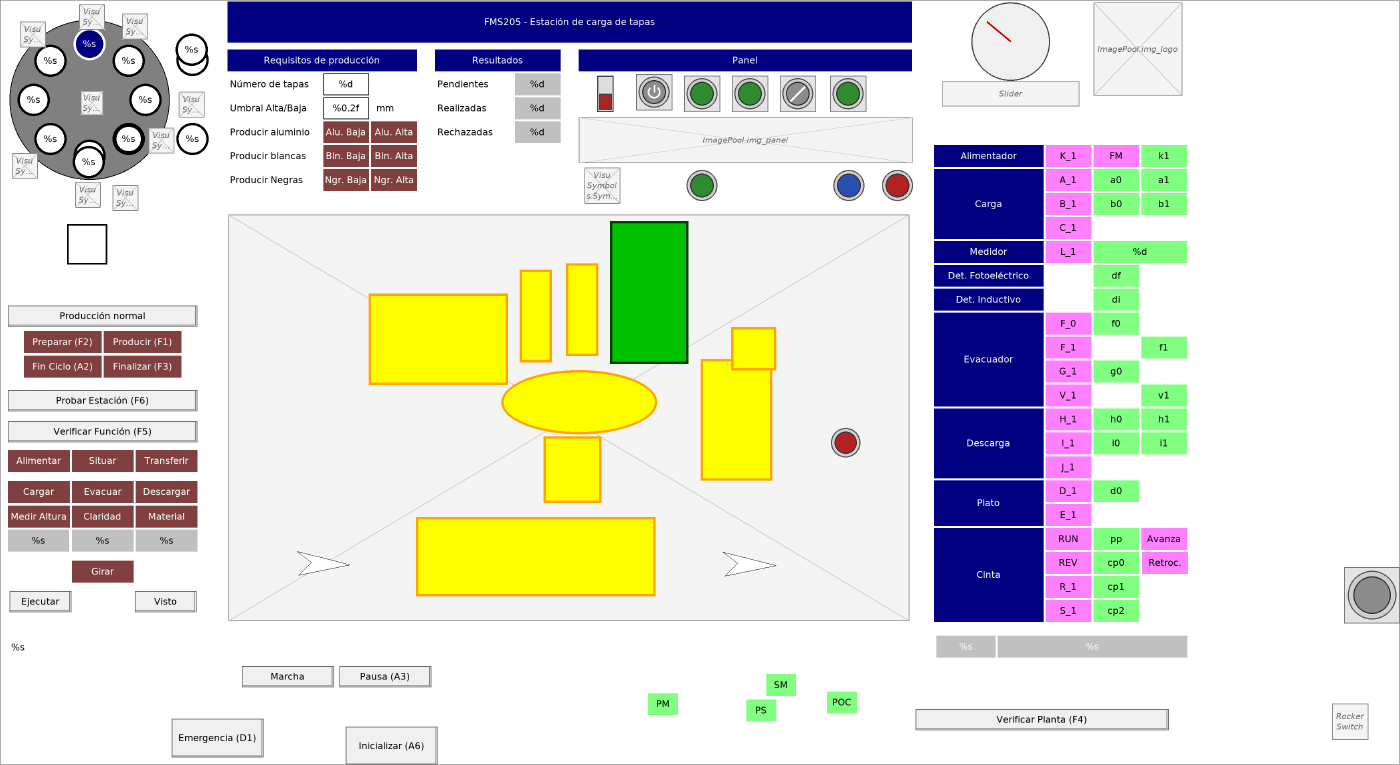
VISUALIZATION L5_FMS205VISU  // 1754x959
    Rectangle (285,2 857x51), "FMS205 - Estación de carga de tapas", colour variable: MAIN.fbFMS205.dr.gmModeColor
        p3450524324: MAIN.fbFMS205.dr.gmModeColor
    Rectangle (285,62 237x27), "Requisitos de producción"
    Rectangle (545,62 157x27), "Resultados"
    Rectangle (725,62 417x27), "Panel"
    Rectangle (285,92 157x27), "Número de tapas"
    Rectangle (405,92 57x27), "%d", text variable: MAIN.fbFMS205.tapas.ReqNumero
        OnMouseClick: write the text variable via VisuDialogs.Numpad, min 1, max 500
    Rectangle (545,92 97x27), "Pendientes"
    Rectangle (645,92 57x27), "%d", text variable: MAIN.fbFMS205.tapas.ResPend
    Rectangle (1036,867 37x27), "POC", input disabled if: NOT MAIN.fbFMS205.dr.gmLocalHost
        toggle MAIN.fbFMS205.fbPanel.hwPOC_PulsadorReset
    Rectangle (812,869 37x27), "PM", input disabled if: NOT MAIN.fbFMS205.dr.gmLocalHost
        toggle MAIN.fbFMS205.fbPanel.hwPM_PulsadorMarcha
    Rectangle (960,845 37x27), "SM", input disabled if: NOT MAIN.fbFMS205.dr.gmLocalHost
        toggle MAIN.fbFMS205.fbPanel.hwSM_SelecAutoManual
    Rectangle (285,122 117x27), "Umbral Alta/Baja"
    Rectangle (405,122 57x27), "%0.2f", text variable: MAIN.fbFMS205.tapas.ReqAlta
        p4168582468: 'Atura en mm mínima para considerar que la tapa es alta'
        OnMouseClick: write the text variable via VisuDialogs.Numpad, min 2, max 5
    Rectangle (465,122 37x27), "mm"
    Rectangle (545,122 117x27), "Realizadas"
    Rectangle (645,122 57x27), "%d", text variable: MAIN.fbFMS205.tapas.ResReal
    Rectangle (285,152 117x27), "Producir aluminio"
    Rectangle (405,152 57x27), "Alu. Baja"
        toggle MAIN.fbFMS205.tapas.ReqAluBaja
    Rectangle (465,152 57x27), "Alu. Alta"
        toggle MAIN.fbFMS205.tapas.ReqAluAlta
    Rectangle (545,152 117x27), "Rechazadas"
    Rectangle (645,152 57x27), "%d", text variable: MAIN.fbFMS205.tapas.ResRech
    Button (1147,889 317x26), "Verificar Planta (F4)", tooltip "%s"
        toggle MAIN.fbFMS205.fbPanel.mdF4Planta
    Rectangle (285,182 117x27), "Producir blancas"
    Rectangle (405,182 57x27), "Bln. Baja"
        toggle MAIN.fbFMS205.tapas.ReqBlnBaja
    Rectangle (465,182 57x27), "Bln. Alta"
        toggle MAIN.fbFMS205.tapas.ReqBlnAlta
    Rectangle (1170,182 137x27), "Alimentador", input disabled if: not MAIN.fbFMS205.dr.cnF4_Planta
    Rectangle (1310,182 57x27), "K_1", input disabled if: not MAIN.fbFMS205.dr.cnF4_Planta
        toggle MAIN.fbFMS205.mdAlimentador.K_1.uiValue
    Rectangle (1370,182 57x27), "FM", input disabled if: not MAIN.fbFMS205.dr.cnF4_Planta
        toggle MAIN.fbFMS205.mdAlimentador.FM.uiValue
    Rectangle (1430,182 57x27), "k1", input disabled if: not MAIN.fbFMS205.dr.cnF4_Planta
        toggle MAIN.fbFMS205.mdAlimentador.k1.uiValue
    Rectangle (285,212 117x27), "Producir Negras"
    Rectangle (405,212 57x27), "Ngr. Baja"
        toggle MAIN.fbFMS205.tapas.ReqNgrBaja
    Rectangle (465,212 57x27), "Ngr. Alta"
        toggle MAIN.fbFMS205.tapas.ReqNgrAlta
    Rectangle (1170,212 137x87), "Carga", input disabled if: not MAIN.fbFMS205.dr.cnF4_Planta
    Rectangle (1310,212 57x27), "A_1", input disabled if: not MAIN.fbFMS205.dr.cnF4_Planta
        toggle MAIN.fbFMS205.mdPickAndPlaceCarga.HOR.uiValue
    Rectangle (1370,212 57x27), "a0", input disabled if: not MAIN.fbFMS205.dr.cnF4_Planta
        toggle MAIN.fbFMS205.mdPickAndPlaceCarga.h0.uiValue
    Rectangle (1430,212 57x27), "a1", input disabled if: not MAIN.fbFMS205.dr.cnF4_Planta
        toggle MAIN.fbFMS205.mdPickAndPlaceCarga.h1.uiValue
    Rectangle (1310,242 57x27), "B_1", input disabled if: not MAIN.fbFMS205.dr.cnF4_Planta
        toggle MAIN.fbFMS205.mdPickAndPlaceCarga.VER.uiValue
    Rectangle (1370,242 57x27), "b0", input disabled if: not MAIN.fbFMS205.dr.cnF4_Planta
        toggle MAIN.fbFMS205.mdPickAndPlaceCarga.v0.uiValue
    Rectangle (1430,242 57x27), "b1", input disabled if: not MAIN.fbFMS205.dr.cnF4_Planta
        toggle MAIN.fbFMS205.mdPickAndPlaceCarga.v1.uiValue
    Rectangle (286,269 837x507), "Estacion"
    Button (303,835 115x26), "Marcha"
        tap MAIN.fbFMS205.fbPanel.swF0_Empezar
    Rectangle (30,415 97x27), "Preparar (F2)", input disabled if: not MAIN.fbFMS205.fbPanel.mdF1Producir
        toggle MAIN.fbFMS205.fbPanel.swF2_Preparar
    Rectangle (130,415 97x27), "Producir (F1)", input disabled if: not MAIN.fbFMS205.fbPanel.mdF1Producir
        toggle MAIN.fbFMS205.fbPanel.swF1_Producir
    Button (215,901 115x48), "Emergencia (D1)", tooltip "%s"
        p4168582468: MAIN.fbFMS205.fbPanel.ttPE_Seta
        toggle MAIN.fbFMS205.fbPanel.swPE_Seta
    Button (425,835 115x26), "Pausa (A3)"
        tap MAIN.fbFMS205.fbPanel.swA3_Estado
    Rectangle (1310,272 57x27), "C_1", input disabled if: not MAIN.fbFMS205.dr.cnF4_Planta
        toggle MAIN.fbFMS205.mdPickAndPlaceCarga.PIN.uiValue
    Rectangle (1170,302 137x27), "Medidor", input disabled if: not MAIN.fbFMS205.dr.cnF4_Planta
    Rectangle (1310,302 57x27), "L_1", input disabled if: not MAIN.fbFMS205.dr.cnF4_Planta
        toggle MAIN.fbFMS205.mdMedidorTapa.L_1.uiValue
    Rectangle (1370,302 117x27), "%d", text variable: MAIN.fbFMS205.mdMedidorTapa.dh, input disabled if: not MAIN.fbFMS205.dr.cnF4_Planta
    Rectangle (1170,332 137x27), "Det. Fotoeléctrico", input disabled if: not MAIN.fbFMS205.dr.cnF4_Planta
    Rectangle (1370,332 57x27), "df", input disabled if: not MAIN.fbFMS205.dr.cnF4_Planta
        toggle MAIN.fbFMS205.mdDetectorFotoelectrico.df.uiValue
    Rectangle (1170,362 137x27), "Det. Inductivo", input disabled if: not MAIN.fbFMS205.dr.cnF4_Planta
    Rectangle (1370,362 57x27), "di", input disabled if: not MAIN.fbFMS205.dr.cnF4_Planta
        toggle MAIN.fbFMS205.mdCaptadorInductivo.di.uiValue
    Rectangle (1170,392 137x117), "Evacuador", input disabled if: not MAIN.fbFMS205.dr.cnF4_Planta
    Rectangle (1310,392 57x27), "F_0", input disabled if: not MAIN.fbFMS205.dr.cnF4_Planta
        toggle MAIN.fbFMS205.mdEvacuador.F_0.uiValue
    Rectangle (1370,392 57x27), "f0", input disabled if: not MAIN.fbFMS205.dr.cnF4_Planta
        toggle MAIN.fbFMS205.mdEvacuador.f0.uiValue
    Button (10,528 237x26), "Verificar Función (F5)", input disabled if: not (MAIN.fbFMS205.dr.gmModeActual=L1_GEMMA.F5VerificacionOrdenada or MAIN.fbFMS205.dr.gmModeActual=L1_GEMMA.A1ParadaInicial)
        toggle MAIN.fbFMS205.fbPanel.mdF5Funcion
    Rectangle (1310,422 57x27), "F_1", input disabled if: not MAIN.fbFMS205.dr.cnF4_Planta
        toggle MAIN.fbFMS205.mdEvacuador.F_1.uiValue
    Rectangle (1430,422 57x27), "f1", input disabled if: not MAIN.fbFMS205.dr.cnF4_Planta
        toggle MAIN.fbFMS205.mdEvacuador.f1.uiValue
    Rectangle (10,564 77x27), "Alimentar", input disabled if: MAIN.fbFMS205.dr.gmModeActual<>L1_GEMMA.F5VerificacionOrdenada
        toggle MAIN.fbFMS205.fbPanel.swF5_Alimentar
    Rectangle (90,703 77x27), "Girar", input disabled if: MAIN.fbFMS205.dr.gmModeActual<>L1_GEMMA.F5VerificacionOrdenada
        toggle MAIN.fbFMS205.fbPanel.swF5_Girar
    Rectangle (90,564 77x27), "Situar", input disabled if: MAIN.fbFMS205.dr.gmModeActual<>L1_GEMMA.F5VerificacionOrdenada
        toggle MAIN.fbFMS205.fbPanel.swF5_Situar
    Rectangle (10,634 77x27), "Medir Altura", input disabled if: MAIN.fbFMS205.dr.gmModeActual<>L1_GEMMA.F5VerificacionOrdenada
        toggle MAIN.fbFMS205.fbPanel.swF5_Medir
    Rectangle (90,634 77x27), "Claridad", input disabled if: MAIN.fbFMS205.dr.gmModeActual<>L1_GEMMA.F5VerificacionOrdenada
        toggle MAIN.fbFMS205.fbPanel.swF5_Claridad
    Rectangle (170,634 77x27), "Material", input disabled if: MAIN.fbFMS205.dr.gmModeActual<>L1_GEMMA.F5VerificacionOrdenada
        toggle MAIN.fbFMS205.fbPanel.swF5_Material
    Rectangle (10,664 76x27), "%s", text variable: MAIN.fbFMS205.mdMedidorTapa.strUi, input disabled if: MAIN.fbFMS205.dr.gmModeActual<>L1_GEMMA.F5VerificacionOrdenada
    Rectangle (90,664 77x27), "%s", text variable: MAIN.fbFMS205.mdDetectorFotoelectrico.strUi, input disabled if: MAIN.fbFMS205.dr.gmModeActual<>L1_GEMMA.F5VerificacionOrdenada
    Rectangle (170,664 77x27), "%s", text variable: MAIN.fbFMS205.mdCaptadorInductivo.strUi, input disabled if: MAIN.fbFMS205.dr.gmModeActual<>L1_GEMMA.F5VerificacionOrdenada
    Rectangle (10,603 77x27), "Cargar", input disabled if: MAIN.fbFMS205.dr.gmModeActual<>L1_GEMMA.F5VerificacionOrdenada
        toggle MAIN.fbFMS205.fbPanel.swF5_Cargar
    Rectangle (90,603 77x27), "Evacuar", input disabled if: MAIN.fbFMS205.dr.gmModeActual<>L1_GEMMA.F5VerificacionOrdenada
        toggle MAIN.fbFMS205.fbPanel.swF5_Evacuar
    Rectangle (170,603 77x27), "Descargar", input disabled if: MAIN.fbFMS205.dr.gmModeActual<>L1_GEMMA.F5VerificacionOrdenada
        toggle MAIN.fbFMS205.fbPanel.swF5_Descargar
    Rectangle (170,564 77x27), "Transferir", input disabled if: MAIN.fbFMS205.dr.gmModeActual<>L1_GEMMA.F5VerificacionOrdenada
        toggle MAIN.fbFMS205.fbPanel.swF5_Transferir
    Button (12,741 77x26), "Ejecutar", input disabled if: MAIN.fbFMS205.dr.gmModeActual<>L1_GEMMA.F5VerificacionOrdenada
        tap MAIN.fbFMS205.fbPanel.swF5_Ejecutar
    Button (169,741 77x26), "Visto", input disabled if: MAIN.fbFMS205.dr.gmModeActual<>L1_GEMMA.F5VerificacionOrdenada
        tap MAIN.fbFMS205.fbPanel.swF5_Ack
    Rectangle (1310,452 57x27), "G_1", input disabled if: not MAIN.fbFMS205.dr.cnF4_Planta
        toggle MAIN.fbFMS205.mdEvacuador.G_1.uiValue
    Rectangle (1370,452 57x27), "g0", input disabled if: not MAIN.fbFMS205.dr.cnF4_Planta
        toggle MAIN.fbFMS205.mdEvacuador.g0.uiValue
    Rectangle (1310,482 57x27), "V_1", input disabled if: not MAIN.fbFMS205.dr.cnF4_Planta
        toggle MAIN.fbFMS205.mdEvacuador.V_1.uiValue
    Rectangle (1430,482 57x27), "v1", input disabled if: not MAIN.fbFMS205.dr.cnF4_Planta
        toggle MAIN.fbFMS205.mdEvacuador.v1.uiValue
    Rectangle (1170,512 137x87), "Descarga", input disabled if: not MAIN.fbFMS205.dr.cnF4_Planta
    Rectangle (1310,512 57x27), "H_1", input disabled if: not MAIN.fbFMS205.dr.cnF4_Planta
        toggle MAIN.fbFMS205.mdPickAndPlaceDescarga.HOR.uiValue
    Rectangle (1370,512 57x27), "h0", input disabled if: not MAIN.fbFMS205.dr.cnF4_Planta
        tap MAIN.fbFMS205.mdPickAndPlaceDescarga.h0.uiValue
        toggle MAIN.fbFMS205.mdPickAndPlaceDescarga.h0.uiValue
    Rectangle (1430,512 57x27), "h1", input disabled if: not MAIN.fbFMS205.dr.cnF4_Planta
        toggle MAIN.fbFMS205.mdPickAndPlaceDescarga.h1.uiValue
    Rectangle (1310,542 57x27), "I_1", input disabled if: not MAIN.fbFMS205.dr.cnF4_Planta
        toggle MAIN.fbFMS205.mdPickAndPlaceDescarga.VER.uiValue
    Rectangle (1370,542 57x27), "i0", input disabled if: not MAIN.fbFMS205.dr.cnF4_Planta
        toggle MAIN.fbFMS205.mdPickAndPlaceDescarga.v0.uiValue
    Rectangle (1430,542 57x27), "i1", input disabled if: not MAIN.fbFMS205.dr.cnF4_Planta
        toggle MAIN.fbFMS205.mdPickAndPlaceDescarga.v1.uiValue
    Rectangle (1310,572 57x27), "J_1", input disabled if: not MAIN.fbFMS205.dr.cnF4_Planta
        toggle MAIN.fbFMS205.mdPickAndPlaceDescarga.PIN.uiValue
    Rectangle (1170,602 137x57), "Plato", input disabled if: not MAIN.fbFMS205.dr.cnF4_Planta
    Rectangle (1310,602 57x27), "D_1", input disabled if: not MAIN.fbFMS205.dr.cnF4_Planta
        toggle MAIN.fbFMS205.mdPlatoDivisor.D_1.uiValue
    Rectangle (1370,602 57x27), "d0", input disabled if: not MAIN.fbFMS205.dr.cnF4_Planta
        toggle MAIN.fbFMS205.mdPlatoDivisor.d0.uiValue
    Rectangle (1310,632 57x27), "E_1", input disabled if: not MAIN.fbFMS205.dr.cnF4_Planta
        toggle MAIN.fbFMS205.mdPlatoDivisor.E_1.uiValue
    Rectangle (1170,662 137x117), "Cinta", input disabled if: not MAIN.fbFMS205.dr.cnF4_Planta
    Rectangle (1310,662 57x27), "RUN", input disabled if: not MAIN.fbFMS205.dr.cnF4_Planta
        toggle MAIN.fbFMS205.mdCinta.RUN.uiValue
    Rectangle (1370,662 57x27), "pp", input disabled if: not MAIN.fbFMS205.dr.cnF4_Planta
        toggle MAIN.fbFMS205.mdCinta.pp.uiValue
    Rectangle (1430,662 57x27), "Avanza", colour toggle: MAIN.fbFMS205.mdCinta.RUN.uiValue and Not MAIN.fbFMS205.mdCinta.REV.uiValue, input disabled if: not MAIN.fbFMS205.dr.cnF4_Planta
        tap MAIN.fbFMS205.fbPanel.swF4_Avanza
    Rectangle (1310,692 57x27), "REV", input disabled if: not MAIN.fbFMS205.dr.cnF4_Planta
        toggle MAIN.fbFMS205.mdCinta.REV.uiValue
    Rectangle (1370,692 57x27), "cp0", input disabled if: not MAIN.fbFMS205.dr.cnF4_Planta
        toggle MAIN.fbFMS205.mdCinta.cp0.uiValue
    Rectangle (1431,692 57x27), "Retroc.", colour toggle: MAIN.fbFMS205.mdCinta.RUN.uiValue and MAIN.fbFMS205.mdCinta.REV.uiValue, input disabled if: not MAIN.fbFMS205.dr.cnF4_Planta
        tap MAIN.fbFMS205.fbPanel.swF4_Retroc
    Rectangle (1310,722 57x27), "R_1", input disabled if: not MAIN.fbFMS205.dr.cnF4_Planta
        toggle MAIN.fbFMS205.mdCinta.R_1.uiValue
    Rectangle (1370,722 57x27), "cp1", input disabled if: not MAIN.fbFMS205.dr.cnF4_Planta
        toggle MAIN.fbFMS205.mdCinta.cp1.uiValue
    Rectangle (1310,752 57x27), "S_1", input disabled if: not MAIN.fbFMS205.dr.cnF4_Planta
        toggle MAIN.fbFMS205.mdCinta.S_1.uiValue
    Rectangle (1370,752 57x27), "cp2", input disabled if: not MAIN.fbFMS205.dr.cnF4_Planta
        toggle MAIN.fbFMS205.mdCinta.cp2.uiValue
    Rectangle (11,798 1117x27), "%s", text variable: main.fbFMS205.fbPanel.swMensaje
    Rectangle (1173,797 74x27), "%s", text variable: MAIN.fbFMS205.fbPanel.gmModeName, colour variable: MAIN.fbFMS205.dr.gmModeColor
        p3450524324: MAIN.fbFMS205.dr.gmModeColor
    Rectangle (1250,797 237x27), "%s", text variable: MAIN.fbFMS205.fbPanel.gmModeDescr, colour variable: MAIN.fbFMS205.dr.gmModeColor
        p3450524324: MAIN.fbFMS205.dr.gmModeColor
    Ellipse (12,25 200x200), colour variable: colVacFrameSin
        p3450524324: colVacFill
    Ellipse (162,105 40x40), "%s", tooltip "%s", text variable: MAIN.fbFMS205.tapas.vstrUi[7], colour variable: MAIN.fbFMS205.tapas.vColorFill[7]
        p2277200375: MAIN.fbFMS205.mdPlatoDivisor.Angulo
        p4168582468: MAIN.fbFMS205.tapas.vstrToolTip[7]
        p55702900: MAIN.fbFMS205.tapas.vColorFont[7]
        p3450524324: MAIN.fbFMS205.tapas.vColorFrame[7]
    Ellipse (141,154 40x40), "%s", tooltip "%s", text variable: MAIN.fbFMS205.tapas.vstrUi[0], colour variable: MAIN.fbFMS205.tapas.vColorFill[0]
        p2277200375: MAIN.fbFMS205.mdPlatoDivisor.Angulo
        p4168582468: MAIN.fbFMS205.tapas.vstrToolTip[0]
        p55702900: MAIN.fbFMS205.tapas.vColorFont[0]
        p3450524324: MAIN.fbFMS205.tapas.vColorFrame[0]
    Ellipse (92,175 40x40), "%s", tooltip "%s", text variable: MAIN.fbFMS205.tapas.vstrUi[1], colour variable: MAIN.fbFMS205.tapas.vColorFill[1]
        p2277200375: MAIN.fbFMS205.mdPlatoDivisor.Angulo
        p4168582468: MAIN.fbFMS205.tapas.vstrToolTip[1]
        p55702900: MAIN.fbFMS205.tapas.vColorFont[1]
        p3450524324: MAIN.fbFMS205.tapas.vColorFrame[1]
    Ellipse (43,154 40x40), "%s", tooltip "%s", text variable: MAIN.fbFMS205.tapas.vstrUi[2], colour variable: MAIN.fbFMS205.tapas.vColorFill[2]
        p2277200375: MAIN.fbFMS205.mdPlatoDivisor.Angulo
        p4168582468: MAIN.fbFMS205.tapas.vstrToolTip[2]
        p55702900: MAIN.fbFMS205.tapas.vColorFont[2]
        p3450524324: MAIN.fbFMS205.tapas.vColorFrame[2]
    Ellipse (22,105 40x40), "%s", tooltip "%s", text variable: MAIN.fbFMS205.tapas.vstrUi[3], colour variable: MAIN.fbFMS205.tapas.vColorFill[3]
        p2277200375: MAIN.fbFMS205.mdPlatoDivisor.Angulo
        p4168582468: MAIN.fbFMS205.tapas.vstrToolTip[3]
        p55702900: MAIN.fbFMS205.tapas.vColorFont[3]
        p3450524324: MAIN.fbFMS205.tapas.vColorFrame[3]
    Ellipse (43,56 40x40), "%s", tooltip "%s", text variable: MAIN.fbFMS205.tapas.vstrUi[4], colour variable: MAIN.fbFMS205.tapas.vColorFill[4]
        p2277200375: MAIN.fbFMS205.mdPlatoDivisor.Angulo
        p4168582468: MAIN.fbFMS205.tapas.vstrToolTip[4]
        p55702900: MAIN.fbFMS205.tapas.vColorFont[4]
        p3450524324: MAIN.fbFMS205.tapas.vColorFrame[4]
    Ellipse (92,35 40x40), "%s", tooltip "%s", text variable: MAIN.fbFMS205.tapas.vstrUi[5], colour variable: MAIN.fbFMS205.tapas.vColorFill[5]
        p2277200375: MAIN.fbFMS205.mdPlatoDivisor.Angulo
        p4168582468: MAIN.fbFMS205.tapas.vstrToolTip[5]
        p55702900: MAIN.fbFMS205.tapas.vColorFont[5]
        p3450524324: MAIN.fbFMS205.tapas.vColorFrame[5]
    Ellipse (141,56 40x40), "%s", tooltip "%s", text variable: MAIN.fbFMS205.tapas.vstrUi[6], colour variable: MAIN.fbFMS205.tapas.vColorFill[6]
        p2277200375: MAIN.fbFMS205.mdPlatoDivisor.Angulo
        p4168582468: MAIN.fbFMS205.tapas.vstrToolTip[6]
        p55702900: MAIN.fbFMS205.tapas.vColorFont[6]
        p3450524324: MAIN.fbFMS205.tapas.vColorFrame[6]
    Image (286,269 853x509), image: ImagePool.img_fms205
    Image (1370,3 111x117), image: ImagePool.img_logo
        p2858320360: sel(MAIN.fbFMS205.dr.gmLocalHost,0,-90)
        OnMouseClick: toggle MAIN.fbFMS205.dr.gmLocalHost
    Image (725,147 418x57), image: ImagePool.img_panel
    Rectangle (935,877 37x27), "PS", input disabled if: NOT MAIN.fbFMS205.dr.gmLocalHost
        toggle MAIN.fbFMS205.fbPanel.hwPS_PulsadorStop
    Image (101,114 28x30), invisible if: MAIN.fbFMS205.mdPlatoDivisor.Ready, image: VisuSymbols.Symbols.ArrowHalfLeftUp
    Image (153,17 32x32), invisible if: MAIN.fbFMS205.mdMedidorTapa.Ready, image: VisuSymbols.Symbols.ArrowBoldDown
    Image (99,5 32x32), invisible if: MAIN.fbFMS205.mdDetectorFotoelectrico.Ready, image: VisuSymbols.Symbols.Download
    Image (25,27 32x32), invisible if: MAIN.fbFMS205.mdCaptadorInductivo.Ready, image: VisuSymbols.Symbols.Download
    Image (15,192 32x32), invisible if: MAIN.fbFMS205.mdEvacuador.Ready, image: VisuSymbols.Symbols.ArrowBoldLeftDown
    Image (94,228 32x32), invisible if: MAIN.fbFMS205.mdPickAndPlaceDescarga.Ready, image: VisuSymbols.Symbols.ArrowBoldDown
    Image (141,232 32x32), invisible if: MAIN.fbFMS205.mdCinta.Ready, image: VisuSymbols.Symbols.ArrowBoldRight
    Meter180 (1171,3 190x98), value: MAIN.fbFMS205.dr.Speed, style: Meter-Meter180-Gray, scale format: %.1f, scale 0..200
    Slider (1180,102 172x31), variable: MAIN.fbFMS205.dr.Speed, scale 1..200
    Rectangle (878,450 89x152), colour variable: MAIN.fbFMS205.mdPickAndPlaceCarga.fbController.colPicFill
        p3450524324: MAIN.fbFMS205.mdPickAndPlaceCarga.fbController.colPicFram
    Button (433,911 115x48), "Inicializar (A6)"
        tap MAIN.fbFMS205.fbPanel.swA6_Inicializar
    Button (10,489 237x26), "Probar Estación (F6)"
        toggle MAIN.fbFMS205.fbPanel.mdF6Probar
    Rectangle (916,410 56x54), angle 322, colour variable: MAIN.fbFMS205.mdAlimentador.fbController.colPicFill
        p3450524324: MAIN.fbFMS205.mdAlimentador.fbController.colPicFram
    Rectangle (764,277 98x179), angle 4, colour variable: MAIN.fbFMS205.mdMedidorTapa.fbController.colPicFill
        p3450524324: MAIN.fbFMS205.mdMedidorTapa.fbController.colPicFram
    Rectangle (709,330 40x116), colour variable: MAIN.fbFMS205.mdDetectorFotoelectrico.fbController.colPicFill
        p3450524324: MAIN.fbFMS205.mdDetectorFotoelectrico.fbController.colPicFram
    Rectangle (651,338 40x116), angle 353, colour variable: MAIN.fbFMS205.mdCaptadorInductivo.fbController.colPicFill
        p3450524324: MAIN.fbFMS205.mdCaptadorInductivo.fbController.colPicFram
    Rectangle (462,368 174x114), angle 351, colour variable: MAIN.fbFMS205.mdEvacuador.fbController.colPicFill
        p3450524324: MAIN.fbFMS205.mdEvacuador.fbController.colPicFram
    Rectangle (681,547 72x83), colour variable: MAIN.fbFMS205.mdPickAndPlaceDescarga.fbController.colPicFill
        p3450524324: MAIN.fbFMS205.mdPickAndPlaceDescarga.fbController.colPicFram
    Rectangle (521,648 300x99), colour variable: MAIN.fbFMS205.mdCinta.fbController.colPicFill
        p3450524324: MAIN.fbFMS205.mdCinta.fbController.colPicFram
    Ellipse (628,464 195x80), colour variable: MAIN.fbFMS205.mdPlatoDivisor.fbController.colPicFill
        p3450524324: MAIN.fbFMS205.mdPlatoDivisor.fbController.colPicFram
    Rectangle (30,446 97x27), angle 359, "Fin Ciclo (A2)", input disabled if: not MAIN.fbFMS205.fbPanel.mdF1Producir
        toggle MAIN.fbFMS205.fbPanel.swA2_FinCiclo
    Rectangle (130,446 97x27), "Finalizar (F3)", input disabled if: not MAIN.fbFMS205.fbPanel.mdF1Producir
        toggle MAIN.fbFMS205.fbPanel.swF3_Finalizar
    Button (10,383 237x26), "Producción normal"
        toggle MAIN.fbFMS205.fbPanel.mdF1Producir
    Polygon (372,691) (372,691) (390,705) (374,721) (438,708), colour variable: MAIN.fbFMS205.mdCinta.colPicFillSituar
        p3450524324: MAIN.fbFMS205.mdCinta.colPicFramSituar
    Polygon (906,692) (906,692) (924,706) (908,722) (972,709), colour variable: MAIN.fbFMS205.mdCinta.colPicFillTransferir
        p3450524324: MAIN.fbFMS205.mdCinta.colPicFramTransferir
    Lamp1 (1032,534 55x42), variable: MAIN.fbFMS205.mdAlimentador.FM.uiValue, style: Lamp-Lamp1-Red
    PowerSwitch (797,93 45x45), tooltip "Conmutador encendido/apagado", variable: MAIN.fbFMS205.fbPanel.hwDPO_DesconectaPO, behaviour: TOGGLE, style: Switch-PowerSwitch-Gray
    DipSwitch (736,95 45x45), tooltip "Parada de emergencia (A1)", variable: MAIN.fbFMS205.fbPanel.swPE_Seta, behaviour: TOGGLE, style: Switch-DipSwitch-Red
    PushSwitch (857,95 45x45), tooltip "Pulsador de marcha", variable: MAIN.fbFMS205.fbPanel.SwPM_PulsadorMarcha, behaviour: TAP, style: Switch-PushSwitch-Green
    PushSwitchLed (1684,711 70x70), behaviour: TOGGLE, style: Switch-PushSwitchLed-Gray
    RockerSwitch (1669,882 45x45), input disabled if: true, behaviour: TOGGLE, style: Switch-RockerSwitch-Red
    RotarySwitch (977,95 45x45), tooltip "Selector manual automático (F4)", variable: MAIN.fbFMS205.fbPanel.swSM_SelecAutoManual, behaviour: TOGGLE, style: Switch-RotarySwitch-Gray
    Ellipse (221,55 40x40), "%s", tooltip "%s", text variable: '???', colour variable: colTapFill
        p4168582468: 'Tapa de altura, claridad y color desconocidos'
        p55702900: colTapFont
        p3450524324: colTapFrameSin
        p2738717112: MAIN.fbFMS205.mdAlimentador.Position
    Ellipse (220,42 40x40), "%s", tooltip "%s", text variable: 'n', colour variable: colTapFill
        p4168582468: 'Cilindro de carga con n tapas'
        p55702900: colTapFont
        p3450524324: colTapFrameSin
    Lamp1 (857,210 45x45), tooltip "Lámpara de marcha", variable: MAIN.fbFMS205.fbPanel.hwLM_LamparaMarcha, style: Lamp-Lamp1-Green
    Lamp1 (1101,210 47x45), tooltip "Lámpara de alarma", variable: MAIN.fbFMS205.fbPanel.hwLA_LamparaAlarma, style: Lamp-Lamp1-Red
    Lamp1 (1040,210 47x45), tooltip "Lámpara de alarma", variable: MAIN.fbFMS205.fbPanel.hwDPO_DesconectaPO, style: Lamp-Lamp1-Blue
    Image (732,210 45x45), tooltip "Avisador sonoro", invisible if: not MAIN.fbFMS205.fbPanel.hwAS_AvisadorSonoro, image: VisuSymbols.Symbols.loudspeakerLoud
    PushSwitch (917,95 45x45), tooltip "Pulsador de parada", variable: MAIN.fbFMS205.fbPanel.swPS_PulsadorStop, behaviour: TAP, style: Switch-PushSwitch-Green
    PushSwitch (1040,95 45x45), tooltip "Pulsador de inicializar (A6)", variable: MAIN.fbFMS205.fbPanel.swPOC_PulsadorReset, behaviour: TAP, style: Switch-PushSwitch-Green
    Ellipse (221,154 40x40), "%s", tooltip "%s", text variable: '???', invisible if: not MAIN.fbFMS205.mdAlimentador._TapaAlimentada, colour variable: colTapFill
        p4168582468: 'Tapa de altura, claridad y color desconocidos'
        p55702900: colTapFont
        p3450524324: colTapFrameSin
        p3560616238: -MAIN.fbFMS205.mdPickAndPlaceCarga.Position
    Rectangle (84,281 50x50)
        p3560616238: MAIN.fbFMS205.mdCinta.Position_Carro
    Image (186,160 32x32), invisible if: MAIN.fbFMS205.mdPickAndPlaceCarga.Ready, image: VisuSymbols.Symbols.ArrowBoldLeft
    Image (224,115 32x32), invisible if: MAIN.fbFMS205.mdAlimentador.Ready, image: VisuSymbols.Symbols.ArrowBoldDown
        p2175578022: MAIN.fbFMS205.mdPickAndPlaceCarga.fbController.colPicFill
    Ellipse (91,183 40x40), "%s", tooltip "%s", text variable: MAIN.fbFMS205.tapas.Desca_strUi, invisible if: MAIN.fbFMS205.mdPickAndPlaceDescarga.Ready, colour variable: MAIN.fbFMS205.tapas.desca_ColorFill
        p4168582468: MAIN.fbFMS205.tapas.Desca_strToolTip
        p55702900: MAIN.fbFMS205.tapas.desca_ColorFont
        p3450524324: MAIN.fbFMS205.tapas.desca_ColorFrame
        p3560616238: MAIN.fbFMS205.mdCinta.Position_Tapa
        p2738717112: MAIN.fbFMS205.mdPickAndPlaceDescarga.Position+MAIN.fbFMS205.mdCinta.PosTapaY
END_VISUALIZATION

(* stored: Version 1.1.0.1, ProductVersion 3.1.4024.11
   Visu L5_FMS205VISU: Id {024cfbd6-56e0-4061-82c5-347b4091fefa} *)
